Staubli VAL3: testMotionCtrl.dtx

mdesc mNomSpeed
public bool bMotionOverrun
public jointRx jJointPos[4]
